(* Logix 5000 project; controller KTC_LAB4 vendor 1 type 14 code 150 rev 30.11; software revision 30.00 *)

TASK MainTask (continuous, watchdog 500 ms) : MainProgram

MODULES
   Local : vendor 1 type 14 code 150 (Compact 0, rev 30.11)
      Counters : Embedded (Compact 3, rev 1.1, Output RPI 20 ms)
      Discrete_IO : Embedded (Compact 1, rev 3.1, Output RPI 20 ms)
      Analog_IO : Embedded (Compact 2, rev 1.1, Output RPI 80 ms)
END_MODULES

PROGRAM MainProgram   (* main routine MainRoutine *)
VAR
   PL0 : ALIAS FOR Local:1:O.Data.0;   // LIGHT 0 NOT A NEVER A
   PL1 : ALIAS FOR Local:1:O.Data.1;   // LIGHT 1 AND
   PL2 : ALIAS FOR Local:1:O.Data.2;   // LIGHT 2 NAND
   PL3 : ALIAS FOR Local:1:O.Data.3;   // LIGHT 3 OR
   PL4 : ALIAS FOR Local:1:O.Data.4;   // LIGHT 4 NOR
   PL5 : ALIAS FOR Local:1:O.Data.5;   // LIGHT 5 XOR
   PL6 : ALIAS FOR Local:1:O.Data.6;   // LIGHT 6 XNOR
   SW4 : ALIAS FOR Local:1:I.Data.4;   // A
   SW5 : ALIAS FOR Local:1:I.Data.5;   // B
END_VAR

ROUTINE MainRoutine   (* ladder *)
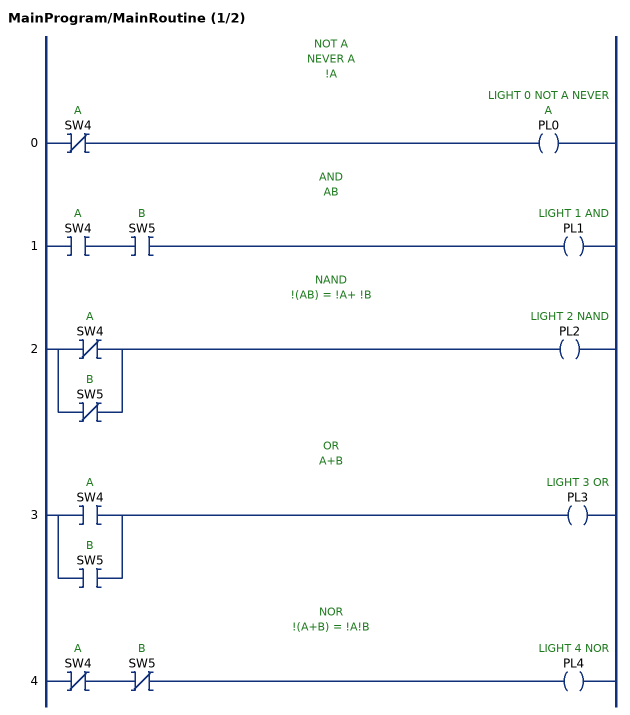
   // NOT A
   // NEVER A
   // !A
   0: XIO(SW4)OTE(PL0);
   // AND
   // AB
   1: XIC(SW4)XIC(SW5)OTE(PL1);
   // NAND
   //  !(AB) = !A+ !B
   2: [XIO(SW4) ,XIO(SW5) ]OTE(PL2);
   // OR
   // A+B
   3: [XIC(SW4) ,XIC(SW5) ]OTE(PL3);
   // NOR
   // !(A+B) = !A!B
   4: XIO(SW4)XIO(SW5)OTE(PL4);
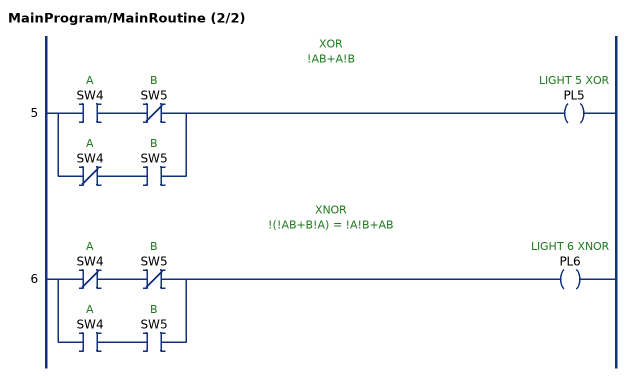
   // XOR
   // !AB+A!B
   5: [XIC(SW4) XIO(SW5) ,XIO(SW4) XIC(SW5) ]OTE(PL5);
   // XNOR
   // !(!AB+B!A) = !A!B+AB
   6: [XIO(SW4) XIO(SW5) ,XIC(SW4) XIC(SW5) ]OTE(PL6);
END_ROUTINE
END_PROGRAM
